// TIA Portal V16 export
// export: Created 2021-07-12T14:47:15.5480904Z, ExportSetting WithDefaults, DisplayName Totally Integrated Automation Portal, DisplayVersion V16, DisplayName TIA Portal Version Control Interface, DisplayVersion V16, DisplayName TIA Portal Openness, DisplayVersion V16, DisplayName STEP 7 Professional, DisplayVersion V16, DisplayName STEP 7 Safety, DisplayVersion V16, DisplayName WinCC Professional, DisplayVersion V16
DATA_BLOCK "InstHydAxisCallFB_Analog2"   // DB33121
{ DB_Accessible_From_OPC_UA := 'FALSE' }
FAMILY : SimaHydTO
VERSION : 1.0
// stored: AutoNumber true, DBAccessibleFromOPCUA false, InstanceOfName LSimaHydTO_HydAxisCall, InstanceOfType FB
"LSimaHydTO_HydAxisCall"
   // VAR_INPUT
   //    axisTO { ExternalAccessible := 'False'; ExternalVisible := 'False'; ExternalWritable := 'False'} : DB_ANY;
   //    pressure_A_RawValue { ExternalAccessible := 'False'; ExternalVisible := 'False'; ExternalWritable := 'False'} : Word;
   //    pressure_B_RawValue { ExternalAccessible := 'False'; ExternalVisible := 'False'; ExternalWritable := 'False'} : Word;
   //    cycleTime { ExternalAccessible := 'False'; ExternalVisible := 'False'; ExternalWritable := 'False'} : UDInt;
   // END_VAR
   // VAR_OUTPUT
   //    error { ExternalAccessible := 'False'; ExternalVisible := 'False'; ExternalWritable := 'False'} : Bool;
   // END_VAR
   // VAR_IN_OUT
   //    axisData : "LSimaHydTO_typeAxisData";
   // END_VAR
   // VAR
   //    statInit { ExternalAccessible := 'False'; ExternalVisible := 'False'; ExternalWritable := 'False'} : Bool;
   //    statTypeOfAxis { ExternalAccessible := 'False'; ExternalVisible := 'False'; ExternalWritable := 'False'} : Int;
   //    instHydAxisFB { ExternalAccessible := 'False'; ExternalVisible := 'False'; ExternalWritable := 'False'; S7_SetPoint := 'True'} : "LSimaHydTO_HydAxis";
   //    instHydSyncAxisFB { ExternalAccessible := 'False'; ExternalVisible := 'False'; ExternalWritable := 'False'; S7_SetPoint := 'True'} : "LSimaHydTO_HydSyncAxis";
   // END_VAR
BEGIN
END_DATA_BLOCK
